(* Schneider Machine Expert - Basic project test4, file version 1.9.0.0 *)
(* ProjectInformations: Name=New project *)

HARDWARE
  Cpu 0: TM221CE16R
  EthernetConfiguration: NetworkName=M221, IpAllocationMode=FixedAddress, IpAddress=0.0.0.0, SubnetMask=0.0.0.0
  SerialLineConfiguration: Baud=Baud19200, Parity=ParityEven, DataBits=DataBits8, StopBits=StopBits1, PhysicalMedium=PhysicalMediumRs485, TransmissionMode=TransmissionModeModbusRtu, SlaveId=1, Addressing=SlaveAddressing
  MastTask: UsePeriodScanMode=false, PeriodScan=100
  FastTask: Period=255
  CpuBehavior: StartingMode=StartAsPreviousState, AutoSaveRamOnEeprom=true, WatchdogPeriod=250

SYMBOLS  (address, symbol, comment, settings)

POU New POU
  (* SectionNumber=1 *)

// Rung 0
  BLK %C0
  LD %I0.0
  R
  LD %I0.1
  S
  LD %I0.2
  CU
  LD %Q0.0
  CD
  OUT_BLK
  LD E
  ST %Q0.0
  LD D
  S %Q0.0
  LD F
  R %Q0.0
  END_BLK
  // as ST:
  //   %C0(R := %I0.0, S := %I0.1, CU := %I0.2, CD := %Q0.0);
  //   %Q0.0 := %C0.E;
  //   IF %C0.D THEN %Q0.0 := TRUE; END_IF;
  //   IF %C0.F THEN %Q0.0 := FALSE; END_IF;
